// TIA Portal V18 export
VAR_GLOBAL   // PLC tag table "RemoteIO_DO_2"
   "oH-shaftLoadingStopperCylinder1_ToWP" AT %Q2000.0 : Bool;   // H-shaft上料线体挡停气缸1_去工作位 / H-shaft上料线体挡停气缸1_去工作位/H-shaft loading line body stops cylinder 1_go to work position
   "oH-shaftLoadingStopperCylinder1_ToHP" AT %Q2000.1 : Bool;   // H-shaft上料线体挡停气缸1_去原始位 / H-shaft上料线体挡停气缸1_去原始位/H-shaft loading line body stops cylinder 1_go to original position
   "oH-shaftLoadingStopperCylinder2_ToWP" AT %Q2000.2 : Bool;   // H-shaft上料线体挡停气缸2_去工作位 / H-shaft上料线体挡停气缸2_去工作位/H-shaft loading line body stops cylinder 2_go to work position
   "oH-shaftLoadingStopperCylinder2_ToHP" AT %Q2000.3 : Bool;   // H-shaft上料线体挡停气缸2_去原始位 / H-shaft上料线体挡停气缸2_去原始位/H-shaft loading line body stops cylinder 2_go to original position
   "oH-shaftLoadingStopperCylinder3_ToWP" AT %Q2000.4 : Bool;   // H-shaft上料线体挡停气缸3_去工作位 / H-shaft上料线体挡停气缸3_去工作位/H-shaft loading line body stops cylinder 3_go to work position
   "oH-shaftLoadingStopperCylinder3_ToHP" AT %Q2000.5 : Bool;   // H-shaft上料线体挡停气缸3_去原始位 / H-shaft上料线体挡停气缸3_去原始位/H-shaft loading line body stops cylinder 3_go to original position
   "oH-shaftLoadingStopperCylinder4_ToWP" AT %Q2000.6 : Bool;   // H-shaft上料线体挡停气缸4_去工作位 / H-shaft上料线体挡停气缸4_去工作位/H-shaft loading line body stops cylinder 4_go to work position
   "oH-shaftLoadingStopperCylinder4_ToHP" AT %Q2000.7 : Bool;   // H-shaft上料线体挡停气缸4_去原始位 / H-shaft上料线体挡停气缸4_去原始位/H-shaft loading line body stops cylinder 4_go to original position
   "oH-shaftTakeStopperCylinder1_ToWP" AT %Q2001.0 : Bool;   // H-shaft取空盘挡停气缸1_去工作位 / H-shaft取空盘挡停气缸1_去工作位/H-shaft takes the empty plate and stops the cylinder 1_go to the working position
   "oH-shaftTakeStopperCylinder1_ToHP" AT %Q2001.1 : Bool;   // H-shaft取空盘挡停气缸1_去原始位 / H-shaft取空盘挡停气缸1_去原始位/H-shaft takes the empty plate and blocks the cylinder 1_go to the original position
   "oH-shaftTakeStopperCylinder2_ToWP" AT %Q2001.2 : Bool;   // H-shaft取空盘挡停气缸2_去工作位 / H-shaft取空盘挡停气缸2_去工作位/H-shaft takes the empty plate and stops the cylinder 2_go to the working position
   "oH-shaftTakeStopperCylinder2_ToHP" AT %Q2001.3 : Bool;   // H-shaft取空盘挡停气缸2_去原始位 / H-shaft取空盘挡停气缸2_去原始位/H-shaft takes the empty plate and blocks the cylinder 2_go to the original position
   "oH-shaftTakeStopperCylinder3_ToWP" AT %Q2001.4 : Bool;   // H-shaft取空盘挡停气缸3_去工作位 / H-shaft取空盘挡停气缸3_去工作位/H-shaft takes the empty plate and stops the cylinder 3_go to the working position
   "oH-shaftTakeStopperCylinder3_ToHP" AT %Q2001.5 : Bool;   // H-shaft取空盘挡停气缸3_去原始位 / H-shaft取空盘挡停气缸3_去原始位/H-shaft takes the empty plate and blocks the cylinder 3_go to the original position
   "RESERVE_Q2001.6" AT %Q2001.6 : Bool;   // 备用_Q2001.6 / 备用_Q2001.6/Standby_Q2001.6
   "RESERVE_Q2001.7" AT %Q2001.7 : Bool;   // 备用_Q2001.7 / 备用_Q2001.7/Standby_Q2001.7
   "oJ-magnetLoadingStopperCylinder1_ToWP" AT %Q2006.0 : Bool;   // J-magnet上料线体挡停气缸1_去工作位 / J-magnet上料线体挡停气缸1_去工作位/J-magnet loading line body stops cylinder 1_go to work position
   "oJ-magnetLoadingStopperCylinder1_ToHP" AT %Q2006.1 : Bool;   // J-magnet上料线体挡停气缸1_去原始位 / J-magnet上料线体挡停气缸1_去原始位/J-magnet loading line body stops cylinder 1_go to original position
   "oJ-magnetLoadingStopperCylinder2_ToWP" AT %Q2006.2 : Bool;   // J-magnet上料线体挡停气缸2_去工作位 / J-magnet上料线体挡停气缸2_去工作位/J-magnet loading line body stops cylinder 2_go to work position
   "oJ-magnetLoadingStopperCylinder2_ToHP" AT %Q2006.3 : Bool;   // J-magnet上料线体挡停气缸2_去原始位 / J-magnet上料线体挡停气缸2_去原始位/J-magnet loading line body stops cylinder 2_go to original position
   "oJ-magnetLoadingStopperCylinder3_ToWP" AT %Q2006.4 : Bool;   // J-magnet上料线体挡停气缸3_去工作位 / J-magnet上料线体挡停气缸3_去工作位/J-magnet loading line body stops cylinder 3_go to work position
   "oJ-magnetLoadingStopperCylinder3_ToHP" AT %Q2006.5 : Bool;   // J-magnet上料线体挡停气缸3_去原始位 / J-magnet上料线体挡停气缸3_去原始位/J-magnet loading line body stops cylinder 3_go to original position
   "oJ-magnetLoadingStopperCylinder4_ToWP" AT %Q2006.6 : Bool;   // J-magnet上料线体挡停气缸4_去工作位 / J-magnet上料线体挡停气缸4_去工作位/J-magnet loading line body stops cylinder 4_go to work position
   "oJ-magnetLoadingStopperCylinder4_ToHP" AT %Q2006.7 : Bool;   // J-magnet上料线体挡停气缸4_去原始位 / J-magnet上料线体挡停气缸4_去原始位/J-magnet loading line body stops cylinder 4_go to original position
   "oJ-magnetTakeStopperCylinder1_ToWP" AT %Q2007.0 : Bool;   // J-magnet取空盘挡停气缸1_去工作位 / J-magnet取空盘挡停气缸1_去工作位/J-magnet takes the empty plate and blocks the cylinder 1_go to the working position
   "oJ-magnetTakeStopperCylinder1_ToHP" AT %Q2007.1 : Bool;   // J-magnet取空盘挡停气缸1_去原始位 / J-magnet取空盘挡停气缸1_去原始位/J-magnet takes the empty plate and blocks the cylinder 1_go to the original position
   "oJ-magnetTakeStopperCylinder2_ToWP" AT %Q2007.2 : Bool;   // J-magnet取空盘挡停气缸2_去工作位 / J-magnet取空盘挡停气缸2_去工作位/J-magnet takes the empty plate and stops the cylinder 2_go to the working position
   "oJ-magnetTakeStopperCylinder2_ToHP" AT %Q2007.3 : Bool;   // J-magnet取空盘挡停气缸2_去原始位 / J-magnet取空盘挡停气缸2_去原始位/J-magnet takes the empty plate and blocks the cylinder 2_go to the original position
   "oJ-magnetTakeStopperCylinder3_ToWP" AT %Q2007.4 : Bool;   // J-magnet取空盘挡停气缸3_去工作位 / J-magnet取空盘挡停气缸3_去工作位/J-magnet takes the empty plate and blocks the cylinder 3_go to the working position
   "oJ-magnetTakeStopperCylinder3_ToHP" AT %Q2007.5 : Bool;   // J-magnet取空盘挡停气缸3_去原始位 / J-magnet取空盘挡停气缸3_去原始位/J-magnet takes the empty plate and blocks the cylinder 3_go to the original position
   "RESERVE_Q2007.6" AT %Q2007.6 : Bool;   // 备用_Q2007.6 / 备用_Q2007.6/Standby_Q2007.6
   "RESERVE_Q2007.7" AT %Q2007.7 : Bool;   // 备用_Q2007.7 / 备用_Q2007.7/Standby_Q2007.7
   "oK-reserveLoadingStopperCylinder1_ToWP" AT %Q2012.0 : Bool;   // K-预留上料线体挡停气缸1_去工作位 / K-预留上料线体挡停气缸1_去工作位/K-reserve the loading line body to stop the cylinder 1_go to the working position
   "oK-reserveLoadingStopperCylinder1_ToHP" AT %Q2012.1 : Bool;   // K-预留上料线体挡停气缸1_去原始位 / K-预留上料线体挡停气缸1_去原始位/K-reserve the loading line body to stop the cylinder 1_go to the original position
   "oK-reserveLoadingStopperCylinder2_ToWP" AT %Q2012.2 : Bool;   // K-预留上料线体挡停气缸2_去工作位 / K-预留上料线体挡停气缸2_去工作位/K-reserve the loading line body to stop the cylinder 2_go to the working position
   "oK-reserveLoadingStopperCylinder2_ToHP" AT %Q2012.3 : Bool;   // K-预留上料线体挡停气缸2_去原始位 / K-预留上料线体挡停气缸2_去原始位/K-reserve the loading line body to stop the cylinder 2_go to the original position
   "oK-reserveLoadingStopperCylinder3_ToWP" AT %Q2012.4 : Bool;   // K-预留上料线体挡停气缸3_去工作位 / K-预留上料线体挡停气缸3_去工作位/K-reserve the loading line body to stop the cylinder 3_go to the working position
   "oK-reserveLoadingStopperCylinder3_ToHP" AT %Q2012.5 : Bool;   // K-预留上料线体挡停气缸3_去原始位 / K-预留上料线体挡停气缸3_去原始位/K-reserve the loading line body to stop the cylinder 3_go to the original position
   "oK-reserveLoadingStopperCylinder4_ToWP" AT %Q2012.6 : Bool;   // K-预留上料线体挡停气缸4_去工作位 / K-预留上料线体挡停气缸4_去工作位/K-reserve the loading line body to stop the cylinder 4_go to the working position
   "oK-reserveLoadingStopperCylinder4_ToHP" AT %Q2012.7 : Bool;   // K-预留上料线体挡停气缸4_去原始位 / K-预留上料线体挡停气缸4_去原始位/K-reserve the loading line body to stop the cylinder 4_go to the original position
   "oK-reserveTakeStopperCylinder1_ToWP" AT %Q2013.0 : Bool;   // K-预留取空盘挡停气缸1_去工作位 / K-预留取空盘挡停气缸1_去工作位/K-reserve empty plate block cylinder 1_go to work position
   "oK-reserveTakeStopperCylinder1_ToHP" AT %Q2013.1 : Bool;   // K-预留取空盘挡停气缸1_去原始位 / K-预留取空盘挡停气缸1_去原始位/K-reserve the empty plate and stop the cylinder 1_go to the original position
   "oK-reserveTakeStopperCylinder2_ToWP" AT %Q2013.2 : Bool;   // K-预留取空盘挡停气缸2_去工作位 / K-预留取空盘挡停气缸2_去工作位/K-reserve empty plate block cylinder 2_go to work position
   "oK-reserveTakeStopperCylinder2_ToHP" AT %Q2013.3 : Bool;   // K-预留取空盘挡停气缸2_去原始位 / K-预留取空盘挡停气缸2_去原始位/K-reserve the empty plate and stop the cylinder 2_go to the original position
   "oK-reserveTakeStopperCylinder3_ToWP" AT %Q2013.4 : Bool;   // K-预留取空盘挡停气缸3_去工作位 / K-预留取空盘挡停气缸3_去工作位/K-reserve empty plate block cylinder 3_go to work position
   "oK-reserveTakeStopperCylinder3_ToHP" AT %Q2013.5 : Bool;   // K-预留取空盘挡停气缸3_去原始位 / K-预留取空盘挡停气缸3_去原始位/K-reserve the empty plate and stop the cylinder 3_go to the original position
   "RESERVE_Q2013.6" AT %Q2013.6 : Bool;   // 备用_Q2013.6 / 备用_Q2013.6/Standby_Q2013.6
   "RESERVE_Q2013.7" AT %Q2013.7 : Bool;   // 备用_Q2013.7 / 备用_Q2013.7/Standby_Q2013.7
   "oL-UnloadingStopperCylinder1_ToWP" AT %Q2018.0 : Bool;   // L-下料线体挡停气缸1_去工作位 / L-下料线体挡停气缸1_去工作位/L-The blanking line body stops the cylinder 1_go to the working position
   "oL-UnloadingStopperCylinder1_ToHP" AT %Q2018.1 : Bool;   // L-下料线体挡停气缸1_去原始位 / L-下料线体挡停气缸1_去原始位/L-The blanking line body stops the cylinder 1_go to the original position
   "oL-UnloadingStopperCylinder2_ToWP" AT %Q2018.2 : Bool;   // L-下料线体挡停气缸2_去工作位 / L-下料线体挡停气缸2_去工作位/L-The blanking line body stops the cylinder 2_go to the working position
   "oL-UnloadingStopperCylinder2_ToHP" AT %Q2018.3 : Bool;   // L-下料线体挡停气缸2_去原始位 / L-下料线体挡停气缸2_去原始位/L-The blanking line body stops the cylinder 2_go to the original position
   "oL-UnloadingStopperCylinder3_ToWP" AT %Q2018.4 : Bool;   // L-下料线体挡停气缸3_去工作位 / L-下料线体挡停气缸3_去工作位/L-The blanking line body stops the cylinder 3_go to the working position
   "oL-UnloadingStopperCylinder3_ToHP" AT %Q2018.5 : Bool;   // L-下料线体挡停气缸3_去原始位 / L-下料线体挡停气缸3_去原始位/L-The blanking line body stops the cylinder 3_go to the original position
   "RESERVE_Q2018.6" AT %Q2018.6 : Bool;   // 备用_Q2018.6 / 备用_Q2018.6/Standby_Q2018.6
   "RESERVE_Q2018.7" AT %Q2018.7 : Bool;   // 备用_Q2018.7 / 备用_Q2018.7/Standby_Q2018.7
END_VAR
